TYPE EtherCAT_Monitor_BatVariables :
STRUCT

	
VaRMS 	:REAL;
VbRMS	:REAL;
VcRMS	:REAL;
IaRMS	:REAL;
IbRMS	:REAL;
IcRMS	:REAL;
Total_ActivePower	:REAL;
Total_ReactivePower	:REAL;
Grid_Frequency	:REAL;
PowerFactor	:REAL;
Vdc	:REAL;
Idc	:REAL;
SoC	:REAL;
SoH	:REAL; 
reserve1: REAL;
reserve2: REAL;

END_STRUCT
END_TYPE

(* stored: Version 1.1.0.1, ProductVersion 3.1.4024.11
   DUT EtherCAT_Monitor_BatVariables: Id {dffeb6dd-77f6-4bd9-85ee-9994cde6b5d4} *)
